Fanuc KAREL source: compact_preamble.KL

PROGRAM KB00190
%NOLOCKGROUP
VAR
P1:REAL;RESULT:REAL
BEGIN
P1=1.0
RESULT=TAN(P1)
END KB00190
